# EPICS autosave request: iocBoot/iocTetrAMM/auto_settings.req
file "quadEM_settings.req",            P=$(P), R=$(R)
file "quadEM_Plugin_settings.req",     P=$(P), R=$(R)
file "commonPlugin_settings.req",      P=$(P), R=$(R)
file "NDStdArrays_settings.req",       P=$(P), R=image1:
